INTERFACE ICUBase

PROPERTY AutomatTask : REFERENCE TO CUBaseAutomat
GET
END_GET
END_PROPERTY

PROPERTY GroundTask : REFERENCE TO CUBaseGround
GET
END_GET
END_PROPERTY

PROPERTY  ManualTask : REFERENCE TO TcoTaskedService
GET
END_GET
END_PROPERTY

PROPERTY ProcessDataManager : REFERENCE TO ProcessDataManager
GET
END_GET
END_PROPERTY

PROPERTY RecoverTask : REFERENCE TO CUBaseRecover
GET
END_GET
END_PROPERTY

PROPERTY StatusInfo :REFERENCE TO CuBaseStatusInfo
GET
END_GET
END_PROPERTY

PROPERTY SuspendTask : REFERENCE TO CUBaseSuspend
GET
END_GET
END_PROPERTY

END_INTERFACE

(* stored: Version 1.1.0.1
   Itf ICUBase: Id {e0435234-64f6-47a6-80fd-c2b672a20857}
   Property AutomatTask: Id {0973134a-28ab-409f-89d6-09a89d3c2b07}
   Get Get: Id {875b00fc-90da-4e77-90bf-2b8bbd7567de}
   Property GroundTask: Id {1d3de518-7983-4b14-bc52-cecc3a9f28ce}
   Get Get: Id {aeb7dbf2-8845-4132-943f-b1517c4d10de}
   Property ManualTask: Id {6e15e50f-dda1-4907-be2f-c73e3cd6490d}
   Get Get: Id {f81b0626-30b3-422b-9427-2ad91ea8af77}
   Property ProcessDataManager: Id {a36eb78f-c57b-4cc6-9daa-ad73e6b1ba37}
   Get Get: Id {7ae5dbe0-0c01-41d7-9272-ab0df9e64885}
   Property RecoverTask: Id {a48486fc-e04e-4a3a-afe9-dac7be323180}
   Get Get: Id {139017a5-85b3-49ae-84ee-9e0279b4115e}
   Property StatusInfo: Id {b09b9df2-c404-481a-a7e9-d29d2da485e5}
   Get Get: Id {f62307e7-aa53-48d1-873d-f1673377d789}
   Property SuspendTask: Id {ad325ad3-fda1-411e-9a82-d90094ec4882}
   Get Get: Id {0f5f179b-9794-4945-8881-f0fe00096457} *)
